FUNCTION CheckAlarm : BOOL

VAR
	thresh : REAL := 90;
	fill : BOOL := GVL.fullness > thresh;
	temp : BOOL := GVL.temp_now > thresh;
END_VAR

CheckAlarm := fill OR temp;

END_FUNCTION

(* stored: Version 1.1.0.1, ProductVersion 3.1.4024.12
   POU CheckAlarm: Id {ce410715-b7c9-458a-8e35-072a529c7159}, SpecialFunc None *)
